FUNCTION_BLOCK StartMotorsProgramAndMovementsTask EXTENDS TcoAbbRoboticsTask
VAR_INPUT
    refStartMotorsAndProgramTask : REFERENCE TO StartMotorsAndProgramTask;
END_VAR
VAR
    _moveParams : TcoAbstractions.TcoRoboticsMovementsParams;
END_VAR
VAR
    _startMotorsAndProgramTask : REFERENCE TO StartMotorsAndProgramTask;
END_VAR

IF NOT __ISVALIDREF(refStartMotorsAndProgramTask) THEN
    Messenger.Post('<#Invalid reference StartMotorAndProgramTask#>', TcoCore.eMessageCategory.ProgrammingError);
    RETURN;
END_IF

_startMotorsAndProgramTask REF= refStartMotorsAndProgramTask;

IF Execute() THEN
    IF _progress = 0 THEN
        IF NOT __ISVALIDREF(inoControl) THEN
            _varInfo := __VARINFO(inoControl);
            Messenger.Programming(_sb.Clear().Append('<#Invalid reference: #>').Append(_varInfo.Symbol).ToString()).Pin();
        ELSIF NOT __ISVALIDREF(inoConfig) THEN
            _varInfo := __VARINFO(inoConfig);
            Messenger.Programming(_sb.Clear().Append('<#Invalid reference: #>').Append(_varInfo.Symbol).ToString()).Pin();
        ELSIF NOT __ISVALIDREF(inoStatus) THEN
            _varInfo := __VARINFO(inoStatus);
            Messenger.Programming(_sb.Clear().Append('<#Invalid reference: #>').Append(_varInfo.Symbol).ToString()).Pin();
        ELSE
            _progress := _progress + 1;
        END_IF
    END_IF

    IF _progress = 1 THEN
        IF _startMotorsAndProgramTask.Invoke().Done THEN
            _progress := _progress + 1;
        END_IF
    END_IF;

    IF _progress = 2 THEN
        inoControl.GlobalSpeed := _moveParams.GlobalSpeed;
        inoControl.ToolNo := _moveParams.ToolNo;
        inoControl.WorkobjectNo := _moveParams.WorkobjectNo;
        inoControl.PointNo := _moveParams.PointNo;
        inoControl.UserSpecSpeed1 := _moveParams.UserSpecSpeed1;
        inoControl.UserSpecSpeed2 := _moveParams.UserSpecSpeed2;
        inoControl.Coordinates := _moveParams.Coordinates;
        inoControl.ActionNo := 254;

        IF inoControl.ActionNo = inoStatus.State.ActionNo THEN
            inoControl.ActionNo := 255;
            _progress := _progress + 1;
        END_IF
    END_IF;

    IF _progress = 3 THEN
        IF inoStatus.State.GlobalSpeed = _moveParams.GlobalSpeed AND
            inoStatus.State.ToolNo = _moveParams.ToolNo AND
            inoStatus.State.WorkobjectNo = _moveParams.WorkobjectNo AND
            inoStatus.State.PointNo = _moveParams.PointNo AND
            inoStatus.State.UserSpecSpeed1 = _moveParams.UserSpecSpeed1 AND
            inoStatus.State.UserSpecSpeed2 = _moveParams.UserSpecSpeed2 AND
            TcoAbstractions.CoordinatesAreEqual(inoStatus.State.Coordinates,
                _moveParams.Coordinates,
                0.01,
                0.01,
                0.01,
                0.01,
                0.01,
                0.01) THEN
            inoControl.ActionNo := 255;
            _progress := _progress + 1;
        END_IF
    END_IF;

    IF _progress = 4 THEN
        IF inoControl.ActionNo = inoStatus.State.ActionNo THEN
            _progress := _progress + 1;
        END_IF
    END_IF;

    IF _progress = 5 THEN
        Messenger.Info(CONCAT('<#Moving to position ID#>: ', INT_TO_STRING(_moveParams.ActionNo)));
        inoControl.ActionNo := _moveParams.ActionNo;

        IF inoControl.ActionNo = inoStatus.State.ActionNo THEN
            inoControl.ActionNo := 255;
            _progress := _progress + 1;
        END_IF
    END_IF;

    IF _progress = 6 THEN
        IF inoControl.ActionNo = inoStatus.State.ActionNo THEN
            DoneWhen(TRUE);
        END_IF
    END_IF;

    CallTimers(TRUE);
    THIS^.ThrowWhen(_errorTimer.Q);
END_IF

IF THIS^.Error AND NOT _errorMessage.Pinned THEN
    THIS^.Restore();
END_IF

METHOD PUBLIC FB_init : BOOL
VAR_INPUT
    bInitRetains : BOOL; // if TRUE, the retain variables are initialized (warm start / cold start)
    bInCopyCode : BOOL; // if TRUE, the instance afterwards gets moved into the copy code (online change)
    ParentObject : ITcoObject;
END_VAR
END_METHOD

METHOD INTERNAL InvokeWithParams : ITcoTaskStatus
VAR_INPUT
    inMoveParams : TcoAbstractions.TcoRoboticsMovementsParams;
END_VAR
_moveParams := inMoveParams;
InvokeWithParams := THIS^.Invoke();
END_METHOD

(*~
    <docu>
        <summary>
            Executes when task is aborted.
        </summary>
    </docu>
~*)
METHOD PROTECTED OnAbort
IF __ISVALIDREF(inoStatus) THEN
    THIS^.inoStatus.ActionDescription := '<#Start motors, program and movements was aborted, while not yet completed!#>';
END_IF;

inoControl.SoftStop := TRUE;
inoControl.QuickStop := FALSE;
END_METHOD

(*~
    <docu>
        <summary>
            Executes when task reaches the ```Done``` state .
        </summary>
    </docu>
~*)
METHOD PROTECTED OnDone
IF __ISVALIDREF(inoStatus) THEN
    THIS^.inoStatus.ActionDescription := '<#Start motors, program and movements finished successfully.#>';
END_IF;

_progress := 0;
END_METHOD

(*~
    <docu>
        <summary>
            Executes when task reaches the ```Error``` state.
        </summary>
    </docu>
~*)
METHOD PROTECTED OnError
VAR
    description : STRING;
END_VAR
description := '<#Start motors, program and movements finished with error.#>';

IF __ISVALIDREF(inoStatus) THEN
    THIS^.inoStatus.ActionDescription := description;
END_IF;

THIS^._errorMessage.Error(_sb.Clear().Append(description).Append(' To restore acknowledge this alarm.').ToString()).Pin();
END_METHOD

METHOD PROTECTED OnStart
IF __ISVALIDREF(inoStatus) THEN
    THIS^.inoStatus.ActionDescription := '<#Start motors, program and movements stared.#>';
END_IF;

CallTimers(FALSE);
inoControl.QuickStop := FALSE;
inoControl.SoftStop := FALSE;
END_METHOD

(*~
    <docu>
        <summary>
            Restores this instance to the Ready state. Can be called explicitly or from within one of the restore mechanisms.
            <para>
                See also <see cref="PlcDocu.TcoCore.TcoTask.AutoRestorable()"/>
            </para>
        </summary>
    </docu>
~*)
METHOD Restore : ITcoRestorable
SUPER^.Restore();
END_METHOD

END_FUNCTION_BLOCK

(* stored: Version 1.1.0.1, ProductVersion 3.1.4024.12
   POU StartMotorsProgramAndMovementsTask: Id {bf97b9ce-c9e3-0f35-1e24-effab0298b12}, SpecialFunc None
   Method FB_init: Id {19a7e90d-7c1d-0040-0877-4edd05388224}
   Method InvokeWithParams: Id {03bb6385-0a25-04a0-08f5-22682b550c9d}
   Method OnAbort: Id {0a7ff24b-6995-0e16-0407-58abe65acaa3}
   Method OnDone: Id {26a4e7c7-cf76-0eb8-0030-5d78190ede54}
   Method OnError: Id {7d9d52fe-07e6-03ba-3423-2c2b9623c945}
   Method OnStart: Id {643539f1-6010-0bad-098f-f9bc81911eb2}
   Method Restore: Id {0c520cf6-de93-04f8-2986-54395f0dffe0} *)
